(* CoDeSys 2.3.9.37 project: Cap5_3.pro *)
(* Libraries: Standard.lib 4.10.05 12:14:46 *)

(* Global variable list: Global_Variables *)
VAR_GLOBAL

(*Entradas*)
	M1: BOOL; (* Pulsador puesta en marcha motor 1 *)
	M2: BOOL; (* Pulsador puesta en marcha motor 2 *)
	M3: BOOL; (* Pulsador puesta en marcha motor 3 *)

	P1: BOOL; (* Pulsador parada motor 1 *)
	P2: BOOL; (* Pulsador parada motor 2*)
	P3: BOOL; (* Pulsador parada motor 3 *)

(*Salidas *)
	Motor1: BOOL;  (*Alimentacion Motor 1 *)
	Motor2: BOOL;  (*Alimentacion Motor 2 *)
	Motor3: BOOL;  (*Alimentacion Motor 3 *)
END_VAR

(* POU PLC_PRG, ST *)
PROGRAM PLC_PRG
VAR

END_VAR

END_PROGRAM

(* Visualisation Botonera
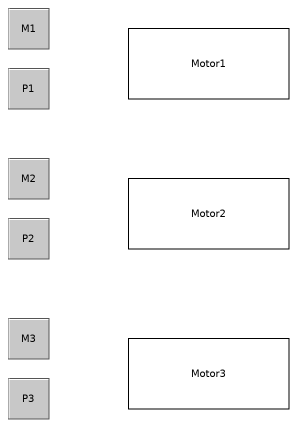
rounded rectangle at (190,50)-(351,121): text "Motor1"; alarm colour if Motor1
button at (70,30)-(111,71): text "M1"; taps M1
button at (70,90)-(111,131): text "P1"; taps P1
rounded rectangle at (190,200)-(351,271): text "Motor2"; alarm colour if Motor2
button at (70,180)-(111,221): text "M2"; taps M2
button at (70,240)-(111,281): text "P2"; taps P2
rounded rectangle at (190,360)-(351,431): text "Motor3"; alarm colour if Motor3
button at (70,340)-(111,381): text "M3"; taps M3
button at (70,400)-(111,441): text "P3"; taps P3
*)
